FUNCTION_BLOCK PusherControl (* Basic Function Block Type *)
  (* Standard: 61499-2 *)
  (* Version 0.0, 1/14/2024, midxav, Template *)
  PACKAGE Main;
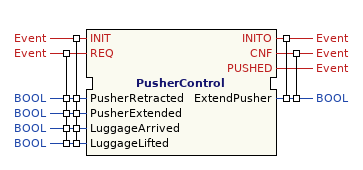
  EVENT_INPUT
    INIT WITH PusherRetracted, PusherExtended, LuggageArrived, LuggageLifted; (* Initialization Request *)
    REQ WITH PusherRetracted, PusherExtended, LuggageArrived, LuggageLifted; (* Normal Execution Request *)
  END_EVENT
  EVENT_OUTPUT
    INITO WITH ExtendPusher; (* Initialization Confirm *)
    CNF WITH ExtendPusher; (* Execution Confirmation *)
    PUSHED;
  END_EVENT
  VAR_INPUT
    PusherRetracted : BOOL;
    PusherExtended : BOOL;
    LuggageArrived : BOOL;
    LuggageLifted : BOOL;
  END_VAR
  VAR_OUTPUT
    ExtendPusher : BOOL;
  END_VAR
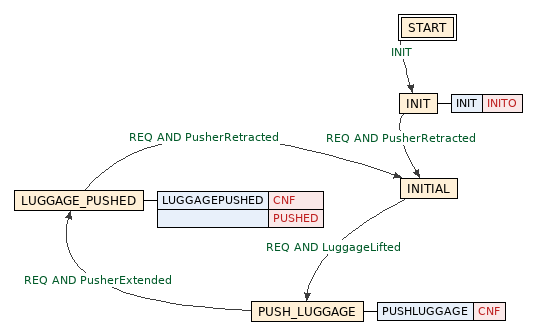
  EC_STATES
    START; (* Initial State *)
    INIT : INIT -> INITO; (* Initialization *)
    INITIAL;
    PUSH_LUGGAGE : PUSHLUGGAGE -> CNF;
    LUGGAGE_PUSHED : LUGGAGEPUSHED -> CNF, -> PUSHED;
  END_STATES
  EC_TRANSITIONS
    START TO INIT := INIT;
    INIT TO INITIAL := REQ AND PusherRetracted;
    PUSH_LUGGAGE TO LUGGAGE_PUSHED := REQ AND PusherExtended;
    LUGGAGE_PUSHED TO INITIAL := REQ AND PusherRetracted;
    INITIAL TO PUSH_LUGGAGE := REQ AND LuggageLifted;
  END_TRANSITIONS
  ALGORITHM INIT IN ST: (* Initialization algorithm *)
ExtendPusher:= FALSE;
  END_ALGORITHM
  ALGORITHM PUSHLUGGAGE IN ST:
ExtendPusher:=TRUE;
  END_ALGORITHM
  ALGORITHM LUGGAGEPUSHED IN ST:
ExtendPusher:=FALSE;
  END_ALGORITHM
END_FUNCTION_BLOCK
